FUNCTION_BLOCK FB_CloseAir
VAR_INPUT
END_VAR
VAR_OUTPUT
END_VAR
VAR
	idx				: INT:=1;
END_VAR


FOR idx:= 1 TO AirNo DO
	AirIsOpen[idx] := FALSE;
END_FOR

END_FUNCTION_BLOCK

(* stored: Version 1.1.0.1, ProductVersion 3.1.4024.9
   POU FB_CloseAir: Id {b107784f-5fa3-429f-b14e-06e0264bdc60}, SpecialFunc None *)
